(* IEC 61131-3 sources: learning-path/06_oop_in_st/exercises/solution/src, 6 files *)

(* ---- ITank.st ---- *)
NAMESPACE FluidHandlingInterfaces
    INTERFACE ITank

        METHOD OpenInlet
        END_METHOD
        METHOD OpenOutlet
        END_METHOD
        METHOD CloseInlet
        END_METHOD
        METHOD CloseOutlet
        END_METHOD

        METHOD Fill
        END_METHOD
        METHOD Flush
        END_METHOD

        METHOD  Close
        END_METHOD

        METHOD Emptying
        END_METHOD

    END_INTERFACE
END_NAMESPACE

(* ---- IValve.st ---- *)
NAMESPACE FluidHandlingClass
    INTERFACE IValve
        METHOD Open
        END_METHOD
        METHOD Close
        END_METHOD
        METHOD GetState : ValveState
        END_METHOD
    END_INTERFACE
END_NAMESPACE

(* ---- basicValve.st ---- *)
NAMESPACE FluidHandlingClass
    CLASS basicValve IMPLEMENTS IValve
        VAR
            _ctrlOpen : BOOL;
            _state : ValveState;
            _isClosed : BOOL;
            _isOpen : BOOL;
        END_VAR

        METHOD PUBLIC Open
            _ctrlOpen := TRUE;
            _isOpen := TRUE;
            _isClosed := FALSE;
        END_METHOD

        METHOD PUBLIC Close
            _ctrlOpen := FALSE;
            _isOpen := FALSE;
            _isClosed := TRUE;
        END_METHOD

        METHOD PUBLIC GetState: FluidHandlingClass.ValveState
            IF (_ctrlOpen) THEN
                GetState := ValveState#Open;
            ELSE
                GetState := ValveState#Closed;
            END_IF;
            _state := GetState;
        END_METHOD

        METHOD PUBLIC WriteCyclic
            VAR_OUTPUT
                ctrlOpen : BOOL;
                isOpen : BOOL;
                isClosed : BOOL;
                state : ValveState;
            END_VAR
            ctrlOpen := _ctrlOpen;
            isOpen := _isOpen;
            isClosed := _isClosed;
            state := _state;
        END_METHOD
    END_CLASS
END_NAMESPACE

(* ---- TankWithShape.st ---- *)
//USING System.Math;
NAMESPACE FluidHandlingInterfaces
    CLASS CylindricalTank EXTENDS TankWithVolume
        VAR PUBLIC
            radium : REAL;
            height : REAL;
        END_VAR
        METHOD VolumeCalculator : REAL
            //volume := TO_REAL(Constants#PI) * radium * radium * height;
            volume := TO_REAL(3.14) * radium * radium * height; // PI is considered Long Real and If I don't change it to real you need to change everything
        END_METHOD
    END_CLASS

    CLASS CubicTank EXTENDS TankWithVolume
        VAR PUBLIC
            side_length : REAL;
        END_VAR
        METHOD VolumeCalculator : REAL
            volume := side_length * side_length * side_length;
        END_METHOD
    END_CLASS
END_NAMESPACE

(* ---- TankWithVolume.st ---- *)
NAMESPACE FluidHandlingInterfaces
    CLASS TankWithVolume IMPLEMENTS ITank
        VAR PUBLIC
            inletValve: IValve;
            outletValve: IValve;
            volume: REAL;
        END_VAR
        VAR PROTECTED
            _capacity : REAL;
            _fill  : BOOL;
            _empty : BOOL;
            _flush : BOOL;
            _close : BOOL;
        END_VAR

        METHOD PUBLIC Capacity : REAL
            VAR_INPUT
                currentVolume : REAL;
            END_VAR
            _capacity := (currentVolume / volume) * 100;
            Capacity := _capacity;
        END_METHOD

        METHOD PUBLIC OpenInlet
            inletValve.Open();
        END_METHOD
        METHOD PUBLIC OpenOutlet
            outletValve.Open();
        END_METHOD
        METHOD PUBLIC CloseInlet
            inletValve.Close();
        END_METHOD
        METHOD PUBLIC CloseOutlet
            outletValve.Close();
        END_METHOD

        METHOD PUBLIC Fill
            this.OpenInlet();
            this.CloseOutlet();
        END_METHOD

        METHOD PUBLIC Flush
            this.OpenInlet();
            this.OpenOutlet();
        END_METHOD

        METHOD PUBLIC Close
            this.CloseInlet();
            this.CloseOutlet();
        END_METHOD

        METHOD PUBLIC Emptying
            this.CloseInlet();
            this.OpenOutlet();
        END_METHOD
        METHOD PUBLIC ReadCyclic
            VAR_INPUT
                Fill : BOOL;
                Empty : BOOL;
                Flush : BOOL;
                Close : BOOL;
            END_VAR
            _fill := Fill;
            _empty := Empty;
            _flush := Flush;
            _close := Close;
        END_METHOD
        METHOD PUBLIC WriteCyclic
            VAR_OUTPUT
                Capacity : REAL;
            END_VAR
            Capacity := _capacity;
        END_METHOD

    END_CLASS
END_NAMESPACE

(* ---- CalculatorWithRegulation.st ---- *)
USING FluidHandlingInterfaces;
USING FluidHandlingClass;
USING System.Timer;

// Imagine that the filling rate is 5 L/s when the inlet valve is Open, so to calculate the maximum filling time: VOLUME TANK/ 5 L/s = TIME FOR TIMER

//CHANGE EVERYTHING FOR REGULATION
PROGRAM CalculatorWithRegulation
    VAR_EXTERNAL
        vInEntry  : ValveWithEntry;
        vOutEntry : ValveWithEntry;
        tankCube : FluidHandlingInterfaces.CubicTank;
        tankCylinder : FluidHandlingInterfaces.CylindricalTank;

        vInCtrlEntry  : BYTE;
        vOutCtrlEntry : BYTE;
        vInRegulator  : BYTE;
        vOutRegulator : BYTE;

        statusInR : ValveState;
        statusOutR : ValveState;

        Close : BOOL;
        Fill  : BOOL;
        Empty : BOOL;
        Flush : BOOL;
        phase : TankState;
    END_VAR
    VAR
        _ton : OnDelay := (duration := T#1s);
        _duration_max : LTIME;
        current_volume : REAL := 0;
        capacity_percentage : REAL;
        _filling_rate : REAL;
        _emptying_rate: REAL;
    END_VAR
    _ton();

    tankCube.VolumeCalculator();

    vInEntry.ReadCyclic(Regulator := TO_REAL(TO_INT(vInRegulator)));
    vOutEntry.ReadCyclic(Regulator := TO_REAL(TO_INT(vOutRegulator)));
    //_duration_max :=  TO_LTIME(TO_LINT(tank.volume / 5));  //Conversion to Time values
    _filling_rate := TO_INT(vInRegulator)/100;
    _emptying_rate := TO_INT(vOutRegulator)/100;
    statusInR := vInEntry.GetState();
    statusOutR := vOutEntry.GetState();

    tankCube.ReadCyclic(Fill := Fill, Empty := Empty, Flush := Flush,  Close := Close);

    CASE phase OF
        //-----------------------------------
        // here's the tank phase close
        //-----------------------------------

            TankState#Close:
            tankCube.Close();
            IF (Fill) THEN
                _ton.signal := TRUE;
                phase := TankState#Filling;
            END_IF;
            IF (Empty) THEN
                _ton.signal := TRUE;
                phase:= TankState#Emptying;
            END_IF;
            IF (Flush) THEN
                _ton.signal := TRUE;
                phase := TankState#Flushing;
            END_IF;
            // next phase after timeout

        //-----------------------------------
        // here's the tank phase Filling
        //-----------------------------------
        TankState#Filling:

            // next phase after timeout
            IF (Fill) THEN
                tankCube.Fill();
                IF (capacity_percentage > 100) THEN
                    _ton.signal := FALSE;
                    phase := TankState#Close;
                END_IF;
                IF _ton.output THEN
                    _ton.signal := FALSE;
                    current_volume := current_volume + 5 *_filling_rate; // Incrementar el volumen en 5 litros por segundo
                    IF current_volume > tankCube.volume THEN
                        current_volume := tankCube.volume; // Asegurar que el volumen no exceda el máximo
                    END_IF;
                    capacity_percentage := (current_volume / tankCube.volume) * 100; // Actualizar el porcentaje de capacidad
                    _ton.signal := TRUE; // Reiniciar el temporizador
                END_IF;

            ELSE
                _ton.signal := FALSE;
                phase := TankState#Close;
            END_IF;
        //-----------------------------------
        // here's the tank phase Emptying
        //-----------------------------------
        TankState#Emptying:
            IF (Empty) THEN
                tankCube.Emptying();
                IF (capacity_percentage <= 0) THEN
                    _ton.signal := FALSE;
                    phase := TankState#Close;
                END_IF;
                IF _ton.output THEN
                    _ton.signal := FALSE;
                    current_volume := current_volume - 5 *_emptying_rate; // Incrementar el volumen en 5 litros por segundo
                    IF current_volume < 0 THEN
                        current_volume := 0; // Asegurar que el volumen no exceda el mínimo
                    END_IF;
                    capacity_percentage := (current_volume / tankCube.volume) * 100; // Actualizar el porcentaje de capacidad
                    _ton.signal := TRUE; // Reiniciar el temporizador
                END_IF;

            ELSE
                _ton.signal := FALSE;
                phase := TankState#Close;
            END_IF;
        //-----------------------------------
        // here's the tank phase Flushing
        //-----------------------------------
        TankState#Flushing:
            IF Flush THEN
                tankCube.Flush();
                _ton.signal := TRUE;
                IF (capacity_percentage <= 0) THEN
                    _ton.signal := FALSE;
                    phase := TankState#Close;
                END_IF;
                IF (capacity_percentage >= 100) THEN
                    _ton.signal := FALSE;
                    phase := TankState#Close;
                END_IF;
                IF _ton.output THEN
                    _ton.signal := FALSE;
                    current_volume := current_volume + 5 * _filling_rate - 5 *_emptying_rate;
                    IF current_volume < 0 THEN
                        current_volume := 0;
                    END_IF;
                    IF current_volume > 100 THEN
                        current_volume := 100;
                    END_IF;
                    capacity_percentage := (current_volume / tankCube.volume) * 100;
                    _ton.signal := TRUE;
                END_IF;
            ELSE
                _ton.signal := FALSE;
                phase := TankState#Close;
            END_IF;
    END_CASE;

    vInEntry.WriteCyclic(ctrlOpen => vInCtrlEntry);
    vOutEntry.WriteCyclic(ctrlOpen => vOutCtrlEntry);
    tankCube.WriteCyclic(Capacity => capacity_percentage);
END_PROGRAM
